{attribute 'linkalways'} 
{attribute 'no_explicit_call' := 'This FB is a CLASS and must be accessed using methods or properties'}
{attribute 'enable_dynamic_creation'}
FUNCTION_BLOCK Node_ContainerType_Vector_Vector_UDINT EXTENDS Node
VAR
    out : _GUID;
END_VAR

METHOD PUBLIC  Clone : I_Node
VAR
	pNode : POINTER TO Node_ContainerType_Vector_Vector_UDINT;
END_VAR
pNode := __NEW(Node_ContainerType_Vector_Vector_UDINT);
Clone := pNode^;
END_METHOD

METHOD FB_init : BOOL
VAR_INPUT
	bInitRetains : BOOL; // if TRUE, the retain variables are initialized (warm start / cold start)
	bInCopyCode : BOOL;  // if TRUE, the instance afterwards gets moved into the copy code (online change)
END_VAR
AddOutput('out', out);
END_METHOD

METHOD PROTECTED OnExecute
out.Value := ContainerType_Vector_Vector_UDINT;
END_METHOD

END_FUNCTION_BLOCK

(* stored: Version 1.1.0.1, ProductVersion 3.1.4026.17
   POU Node_ContainerType_Vector_Vector_UDINT: Id {2d7d338f-eb1e-040a-022f-72f730c7f959}, SpecialFunc None
   Folder Constructor: Id {0d4c9142-7024-0831-0826-395ec07193df}
   Method Clone: Id {e0ef5721-3121-0680-217b-950b782811fa}
   Method FB_init: Id {42b37653-cb05-00d7-0156-f3aae2ff0632}
   Method OnExecute: Id {96bdaa0e-b80b-09ed-34be-2b3d510c5e6d} *)
